// SIMATIC S7-200 project (STEP 7-Micro/WIN), CPU 224XP REL 02.01

SYMBOL_TABLE USUARIO1
P_PLANTA_B       I0.0
P_CABINA_B       I0.1
P_PLANTA_1       I0.2
P_CABINA_1       I0.3
FC_PLANTA_BAJA   I0.4
FC_PLANTA_1      I0.5
S_L_U1V1W1_RST   Q0.0
S_R_U2V2W2_RST   Q0.1
CORTOCIRQUITADO_SB Q0.2
B_L_U1V1W1_SRT   Q0.3
B_R_U2V2W2_SRT   Q0.4
END_SYMBOL_TABLE

ORGANIZATION_BLOCK PRINCIPAL:OB1
TITLE=COMENTARIOS DEL PROGRAMA
BEGIN
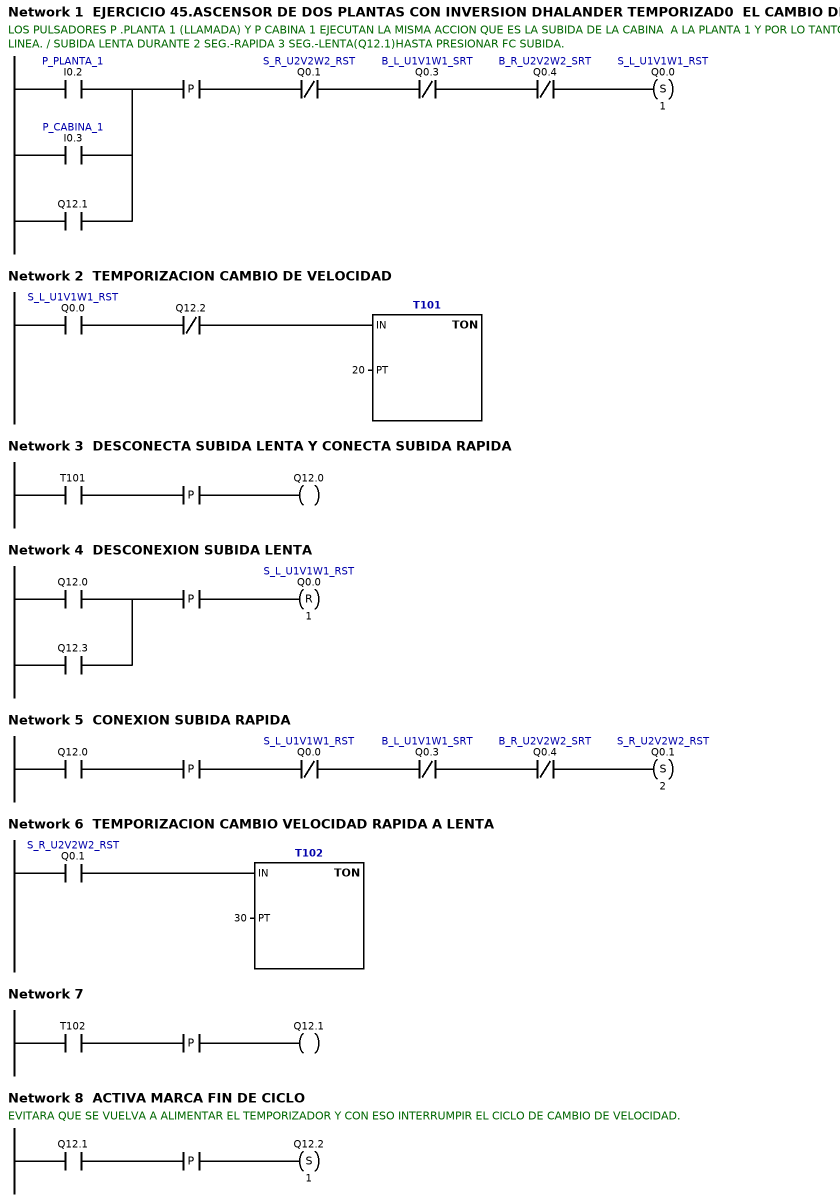
Network 1 // EJERCICIO 45.ASCENSOR DE DOS PLANTAS CON INVERSION DHALANDER TEMPORIZAD0  EL CAMBIO DE VELOCIDAD TANTO SUBIDA COMO BAJADA.
// LOS PULSADORES P .PLANTA 1 (LLAMADA) Y P CABINA 1 EJECUTAN LA MISMA ACCION QUE ES LA SUBIDA DE LA CABINA  A LA PLANTA 1 Y POR LO TANTO SE PTOGRAMAN EN PARALELO EN LA MISMA LINEA.
// SUBIDA LENTA DURANTE 2 SEG.-RAPIDA 3 SEG.-LENTA(Q12.1)HASTA PRESIONAR FC SUBIDA.
LD     P_PLANTA_1:I0.2
O      P_CABINA_1:I0.3
O      Q12.1
EU
AN     S_R_U2V2W2_RST:Q0.1
AN     B_L_U1V1W1_SRT:Q0.3
AN     B_R_U2V2W2_SRT:Q0.4
S      S_L_U1V1W1_RST:Q0.0, 1
Network 2 // TEMPORIZACION CAMBIO DE VELOCIDAD
LD     S_L_U1V1W1_RST:Q0.0
AN     Q12.2
TON    T101, 20
Network 3 // DESCONECTA SUBIDA LENTA Y CONECTA SUBIDA RAPIDA
LD     T101
EU
=      Q12.0
Network 4 // DESCONEXION SUBIDA LENTA
LD     Q12.0
O      Q12.3
EU
R      S_L_U1V1W1_RST:Q0.0, 1
Network 5 // CONEXION SUBIDA RAPIDA
LD     Q12.0
EU
AN     S_L_U1V1W1_RST:Q0.0
AN     B_L_U1V1W1_SRT:Q0.3
AN     B_R_U2V2W2_SRT:Q0.4
S      S_R_U2V2W2_RST:Q0.1, 2
Network 6 // TEMPORIZACION CAMBIO VELOCIDAD RAPIDA A LENTA 
LD     S_R_U2V2W2_RST:Q0.1
TON    T102, 30
Network 7
LD     T102
EU
=      Q12.1
Network 8 // ACTIVA MARCA FIN DE CICLO
// EVITARA QUE SE VUELVA A ALIMENTAR EL TEMPORIZADOR Y CON ESO INTERRUMPIR EL CICLO DE CAMBIO DE VELOCIDAD.
LD     Q12.1
EU
S      Q12.2, 1
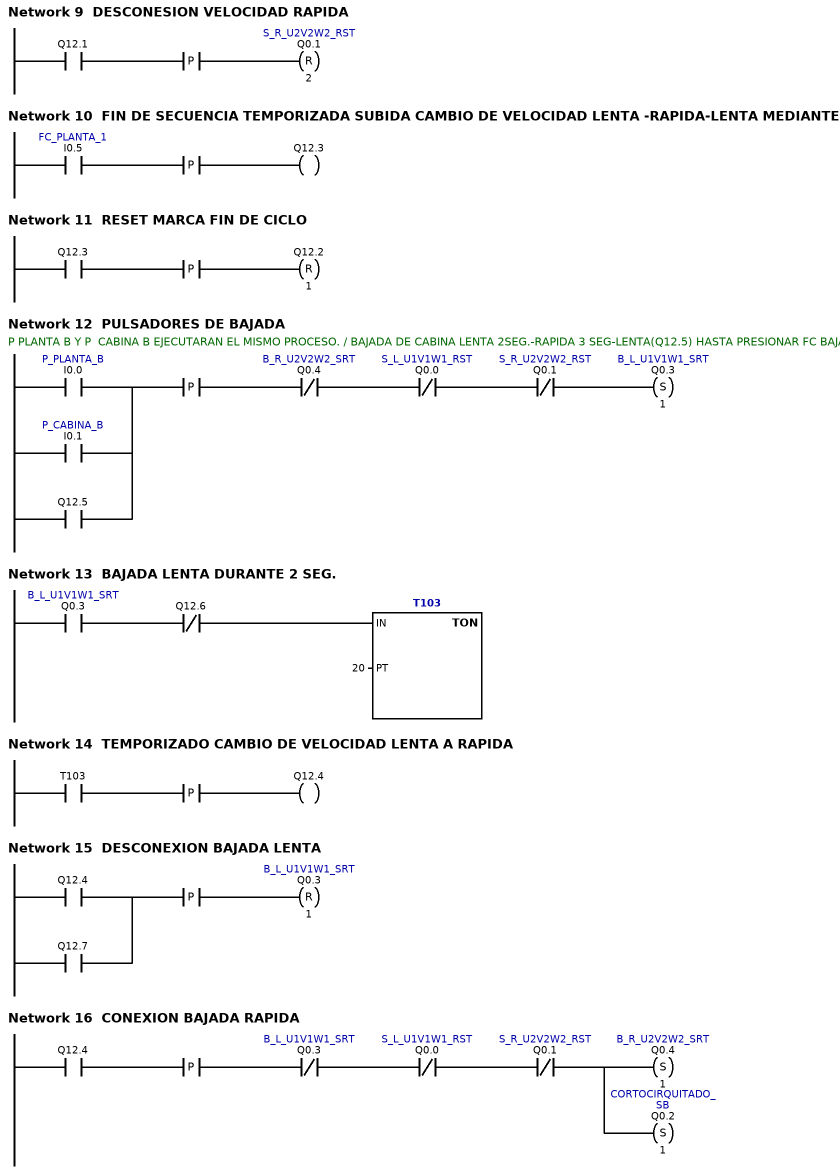
Network 9 // DESCONESION VELOCIDAD RAPIDA
LD     Q12.1
EU
R      S_R_U2V2W2_RST:Q0.1, 2
Network 10 // FIN DE SECUENCIA TEMPORIZADA SUBIDA CAMBIO DE VELOCIDAD LENTA -RAPIDA-LENTA MEDIANTE FC CARRERA PLANTA 1.
LD     FC_PLANTA_1:I0.5
EU
=      Q12.3
Network 11 // RESET MARCA FIN DE CICLO
LD     Q12.3
EU
R      Q12.2, 1
Network 12 // PULSADORES DE BAJADA
// P PLANTA B Y P  CABINA B EJECUTARAN EL MISMO PROCESO.
// BAJADA DE CABINA LENTA 2SEG.-RAPIDA 3 SEG-LENTA(Q12.5) HASTA PRESIONAR FC BAJADA.
LD     P_PLANTA_B:I0.0
O      P_CABINA_B:I0.1
O      Q12.5
EU
AN     B_R_U2V2W2_SRT:Q0.4
AN     S_L_U1V1W1_RST:Q0.0
AN     S_R_U2V2W2_RST:Q0.1
S      B_L_U1V1W1_SRT:Q0.3, 1
Network 13 // BAJADA LENTA DURANTE 2 SEG.
LD     B_L_U1V1W1_SRT:Q0.3
AN     Q12.6
TON    T103, 20
Network 14 // TEMPORIZADO CAMBIO DE VELOCIDAD LENTA A RAPIDA
LD     T103
EU
=      Q12.4
Network 15 // DESCONEXION BAJADA LENTA 
LD     Q12.4
O      Q12.7
EU
R      B_L_U1V1W1_SRT:Q0.3, 1
Network 16 // CONEXION BAJADA RAPIDA
LD     Q12.4
EU
AN     B_L_U1V1W1_SRT:Q0.3
AN     S_L_U1V1W1_RST:Q0.0
AN     S_R_U2V2W2_RST:Q0.1
S      B_R_U2V2W2_SRT:Q0.4, 1
S      CORTOCIRQUITADO_SB:Q0.2, 1
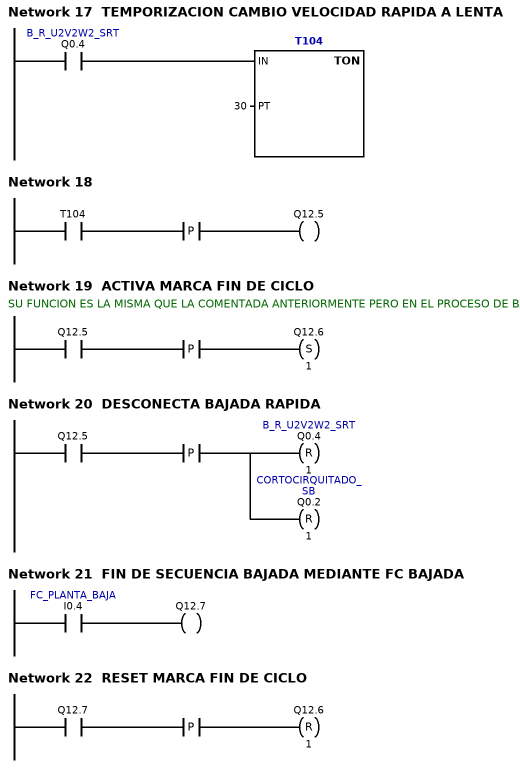
Network 17 // TEMPORIZACION CAMBIO VELOCIDAD RAPIDA A LENTA 
LD     B_R_U2V2W2_SRT:Q0.4
TON    T104, 30
Network 18
LD     T104
EU
=      Q12.5
Network 19 // ACTIVA MARCA FIN DE CICLO 
// SU FUNCION ES LA MISMA QUE LA COMENTADA ANTERIORMENTE PERO EN EL PROCESO DE BAJADA.
LD     Q12.5
EU
S      Q12.6, 1
Network 20 // DESCONECTA BAJADA RAPIDA 
LD     Q12.5
EU
R      B_R_U2V2W2_SRT:Q0.4, 1
R      CORTOCIRQUITADO_SB:Q0.2, 1
Network 21 // FIN DE SECUENCIA BAJADA MEDIANTE FC BAJADA
LD     FC_PLANTA_BAJA:I0.4
=      Q12.7
Network 22 // RESET MARCA FIN DE CICLO
LD     Q12.7
EU
R      Q12.6, 1
END_ORGANIZATION_BLOCK
